KUKA KRL program: weld.src, weld.dat

--- weld.src ---
&ACCESS RVO1
&REL 1
&PARAM DISKPATH = KRC:\R1\Program\Production
DEF weld( )
   DECL INT contID	; ContainerID
   DECL BOOL RSI_ON
   ;FOLD INI;%{PE}
      ;FOLD BASISTECH INI
         GLOBAL INTERRUPT DECL 3 WHEN $STOPMESS==TRUE DO IR_STOPM ( )
         INTERRUPT DECL 5 WHEN VIS_HEIGHT == VIS_HEIGHT_NOT_IN_RANGE DO DisableRSI()
         INTERRUPT ON 3
         BAS (#INITMOV,0 )
      ;ENDFOLD (BASISTECH INI)
      ;FOLD USER INI
         ;Make your modifications here

      ;ENDFOLD (USER INI)
   ;ENDFOLD (INI)

   Xdummy_point = $POS_ACT
   PTP Xdummy_point

   ; find the seam (min of 2 tracks)
   counter = 0
   WHILE (counter < minCount) OR (TrackSeam()==FALSE)
      counter = counter + 1
   ENDWHILE

   ;FOLD HandShake[25 : Wait for table position], WAIT on Response
      HandShake_Set (25,false)
      HandShake_Check (25,false)
   ;ENDFOLD

   WHILE weldActive
      throwawaybool = TrackSeam()

      if RSI_GO_MANUAL== FALSE then
         RSI_ON = RSI_SetUp_TurnOn(RSI_ID)
         ; DisableRSI_Pos()

         $SEN_PINT[RSI_MoveCorr_Stop]=1
         RSI_MOVECORR()

         RSI_RESET_PIDS()
         TurnOffRSI(RSI_ID)
         Xdummy_point = $POS_ACT
         PTP Xdummy_point
      ENDIF
   ENDWHILE

   BAS(#TOOL, 1) ; select first tool
   BAS(#BASE, 1) ; select base 1
   BAS(#VEL_CP, 0.050) ; m/s
   BAS(#ACC_CP, 50) ; use max acceleration


   LIN_REL { Z -50 } #TOOL

   HomePos()

   Exit_Program()

END

--- weld.dat ---
&ACCESS RVO1
&REL 1
&PARAM DISKPATH = KRC:\R1\Program\Production
DEFDAT  weld
;FOLD EXTERNAL DECLARATIONS;%{PE}%MKUKATPBASIS,%CEXT,%VCOMMON,%P
;FOLD BASISTECH EXT;%{PE}%MKUKATPBASIS,%CEXT,%VEXT,%P
EXT  BAS (BAS_COMMAND  :IN,REAL  :IN )
;ENDFOLD (BASISTECH EXT)
;FOLD USER EXT;%{E}%MKUKATPUSER,%CEXT,%VEXT,%P
;Make your modifications here
;ENDFOLD (USER EXT)
;ENDFOLD (EXTERNAL DECLARATIONS)

DECL BOOL throwawaybool

DECL INT nType
DECL INT counter=2
DECL INT minCount=2

DECL BASIS_SUGG_T LAST_BASIS={POINT1[] "P1                      ",POINT2[] "P1                      ",CP_PARAMS[] "CPDAT0                  ",PTP_PARAMS[] "PDAT1                   ",CONT[] "                        ",CP_VEL[] "2.0                     ",PTP_VEL[] "20                      ",SYNC_PARAMS[] "SYNCDAT                 ",SPL_NAME[] "S0                      ",A_PARAMS[] "ADAT0                   "}
DECL E6POS XP1={X 403.077454,Y 1348.19373,Z 1142.98474,A -164.725662,B -89.6085281,C 100.191284,S 6,T 51,E1 0.0,E2 0.0,E3 0.0,E4 0.0,E5 0.0,E6 0.0}
DECL FDAT FP1={TOOL_NO 1,BASE_NO 0,IPO_FRAME #BASE,POINT2[] " ",TQ_STATE FALSE}
DECL PDAT PPDAT1={VEL 100.000,ACC 5.00000,APO_DIST 100.000,APO_MODE #CDIS,GEAR_JERK 50.0000,EXAX_IGN 0}
ENDDAT
